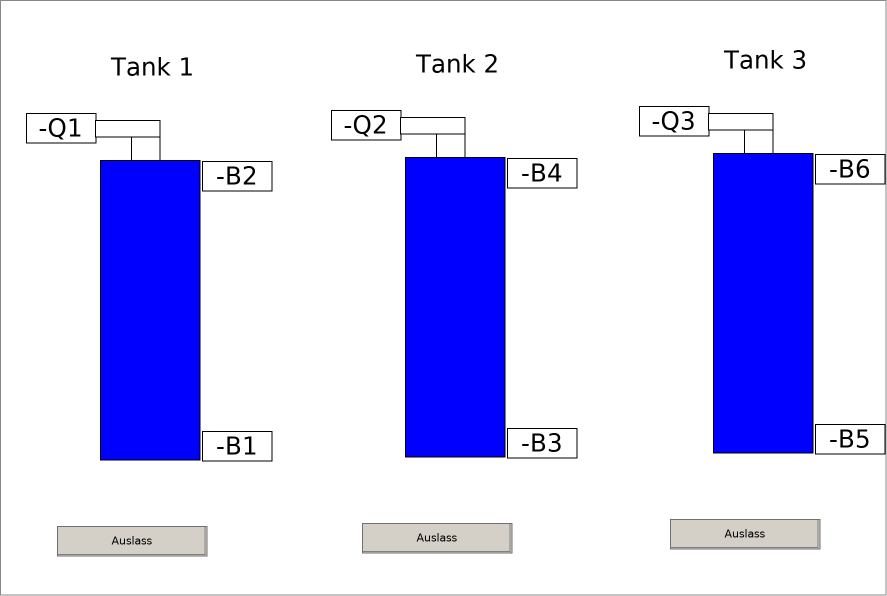
VISUALIZATION TankFuellAnlage  // 887x596
    Rectangle (128,461 29x133), colour toggle: MAIN.Simulation.xAuslass1
    Rectangle (131,120 29x305), colour toggle: DIO.Q1
    Rectangle (100,160 100x300)
    Rectangle (100,160 100x300)
        p2773130477: MAIN.Simulation.uiFuellstandTank1
    Label (105,52 95x30), "Tank 1"
    Button (57,526 150x30), "Auslass"
        tap MAIN.Simulation.xAuslass1
    Rectangle (202,161 70x30), "-B2", colour toggle: VISU.B2
    Rectangle (202,431 70x30), "-B1", colour toggle: VISU.B1
    Rectangle (26,113 70x30), "-Q1", colour toggle: DIO.Q1
    Rectangle (95,120 65x17), colour toggle: DIO.Q1
    Rectangle (436,117 29x305), colour toggle: DIO.Q2
    Rectangle (405,157 100x300)
    Rectangle (405,157 100x300)
        p2773130477: MAIN.Simulation.uiFuellstandTank2
    Label (410,49 95x30), "Tank 2"
    Button (362,523 150x30), "Auslass"
        tap MAIN.Simulation.xAuslass2
    Rectangle (507,158 70x30), "-B4", colour toggle: VISU.B4
    Rectangle (507,428 70x30), "-B3", colour toggle: VISU.B3
    Rectangle (331,110 70x30), "-Q2", colour toggle: DIO.Q2
    Rectangle (400,117 65x17), colour toggle: DIO.Q2
    Rectangle (391,183 29x301), colour toggle: DIO.Q1
    Rectangle (744,113 29x305), colour toggle: DIO.Q3
    Rectangle (713,153 100x300)
    Rectangle (713,153 100x300)
        p2773130477: MAIN.Simulation.uiFuellstandTank3
    Label (718,45 95x30), "Tank 3"
    Button (670,519 150x30), "Auslass"
        tap MAIN.Simulation.xAuslass3
    Rectangle (815,154 70x30), "-B6", colour toggle: VISU.B6
    Rectangle (815,424 70x30), "-B5", colour toggle: VISU.B5
    Rectangle (639,106 70x30), "-Q3", colour toggle: DIO.Q3
    Rectangle (708,113 65x17), colour toggle: DIO.Q3
    Rectangle (699,179 29x301), colour toggle: DIO.Q1
    Rectangle (132,150 29x305), colour toggle: DIO.Q1
    Rectangle (436,151 29x305), colour toggle: DIO.Q2
    Rectangle (747,151 29x305), colour toggle: DIO.Q3
    Rectangle (437,458 29x133), colour toggle: MAIN.Simulation.xAuslass2
    Rectangle (749,455 29x133), colour toggle: MAIN.Simulation.xAuslass3
END_VISUALIZATION

(* stored: Version 1.1.0.1, ProductVersion 3.1.4022.6
   Visu TankFuellAnlage: Id {116ef40b-496c-489a-a025-1af3552c8f1e} *)
